FUNCTION_BLOCK IO_READER
  (* Standard: 61499-2 *)
  (* Version 11-01-12, GASR *)
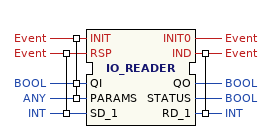
  EVENT_INPUT
    INIT WITH QI, PARAMS;
    RSP WITH SD_1;
  END_EVENT
  EVENT_OUTPUT
    INIT0;
    IND WITH RD_1;
  END_EVENT
  VAR_INPUT
    QI : BOOL;
    PARAMS : ANY;
    SD_1 : INT;
  END_VAR
  VAR_OUTPUT
    QO : BOOL;
    STATUS : BOOL;
    RD_1 : INT;
  END_VAR
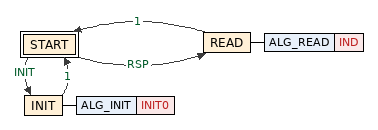
  EC_STATES
    START;
    READ : ALG_READ -> IND;
    INIT : ALG_INIT -> INIT0;
  END_STATES
  EC_TRANSITIONS
    START TO INIT := INIT;
    INIT TO START := 1;
    START TO READ := RSP;
    READ TO START := 1;
  END_TRANSITIONS
  ALGORITHM ALG_INIT IN Lua:

  END_ALGORITHM
  ALGORITHM ALG_READ IN Lua:
RD_1 := GET_REG(SD_1);
  END_ALGORITHM
END_FUNCTION_BLOCK
